// TIA Portal V20 export
// export: Created 2025-12-01T14:56:17.9441989Z, ExportSetting None, DisplayName Totally Integrated Automation Portal, DisplayVersion V20 Update 3, DisplayName TIA Portal Openness, DisplayVersion V20 Update 3, DisplayName TIA Portal Version Control Interface, DisplayVersion V20 Update 3, DisplayName STEP 7 Professional, DisplayVersion V20 Update 3, DisplayName STEP 7 Safety, DisplayVersion V20 Update 2, DisplayName WinCC Basic/Comfort/Advanced, DisplayVersion V20 Update 3, DisplayName WinCC Professional, DisplayVersion V20 Update 3, DisplayName WinCC Unified, DisplayVersion V20 Update 3
TYPE "Avisos_HMI_Mesa"
   STRUCT
      SiguientePosUT : Bool;
      AnteriorPosUT : Bool;
      Bit_02 : Bool;
      Bit_03 : Bool;
      PeticionVisualizarMesa : Bool;
      Bit_05 : Bool;
      Bit_06 : Bool;
      Bit_07 : Bool;
      CambiarUT_SiguientePosUT : Bool;
      CambiarUT_AnteriorPosUT : Bool;
      CambiarUT_DeMesa : Bool;
      Eliminar_UT : Bool;
      Crear_UT : Bool;   // Crear una Nueva UT en la Mesa (Mckey = 0)
      Bit_15 : Bool;
      Bit_16 : Bool;
      KeepAlive : Bool;
   END_STRUCT;
END_TYPE
